# EPICS autosave request: iocBoot/ioc13lab2/auto_settings.req
file "Keithley2kDMM_mf10_settings.req", P=13LAB2:, Dmm=DMM1
file "scan_settings.req", P=13LAB2:, S=scan1
file "scan_settings.req", P=13LAB2:, S=scan2
file "scan_settings.req", P=13LAB2:, S=scan3
file "scan_settings.req", P=13LAB2:, S=scan4
file "CARS_8_motor_settings.req", P=13LAB2:
